// TIA Portal V20 export
FUNCTION "FC_Utilities" : Void   // FC1, SCL
{ S7_Optimized_Access := 'TRUE' }
// stored: SetENOAutomatically false
   VAR_INPUT
      rInput : Real;
      rMin : Real;
      rMax : Real;
   END_VAR
   VAR_OUTPUT
      rResult : Real;
   END_VAR
BEGIN

   #rResult := (#rInput * (#rMax - #rMin)) + #rMin;
END_FUNCTION
